// SIMATIC S7-200 SMART project (STEP 7-Micro/WIN SMART), CPU ST20

SYMBOL_TABLE Table 1
Counter_1        C1
Counted          VW0
CTRL_Done        M0.0
MSG_Done_0       M0.1
MSG_Done_1       M0.2
Error_0          MB1
Error_1          MB2
Error_2          MB3
MSG_0            M4.0
MSG_1            M4.1
TmpBit           M4.2
END_SYMBOL_TABLE

SYMBOL_TABLE System Symbols
Always_On        SM0.0    // Always ON
END_SYMBOL_TABLE

ORGANIZATION_BLOCK MAIN:OB1
TITLE=Program Comments
BEGIN
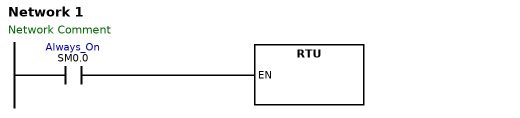
Network 1
// Network Comment
LD     Always_On:SM0.0
CALL   RTU:SBR10
END_ORGANIZATION_BLOCK

// SBR0: protected block, not included

// SBR1: protected block, not included

// SBR2: protected block, not included
